(* Logix 5000 project; controller HaileeRenkersACIM5030ProjectFinalVersion vendor 1 type 14 code 54 rev 20.12; software revision 20.01 *)

TASK MainTask (continuous, watchdog 500 ms) : MainProgram

MODULES
   Local : vendor 1 type 14 code 54 (ICP 0, rev 20.12)
      DCinputmodule : 1756-IB16 (ICP 1, rev 3.3, Input RPI 20 ms)   // inputmodule for discrete dc inputs
      outputrelay : 1756-OW16I (ICP 2, rev 3.2, Output RPI 20 ms)   // outputrelay
      inputcardslot3 : 1756-IF8 (ICP 3, rev 1.5, Input RPI 100 ms)
      highspeedcounter : 1756-HSC (ICP 6, rev 3.4, Output RPI 2 ms)
      Ethernet : 1756-ENBT (ICP 7, Ethernet 142.232.195.220, rev 4.8)
         Powerflex : vendor 1 type 123 code 50 (Ethernet 142.232.195.234, rev 5.1, Output RPI 20 ms)
             : vendor 1 type 123 code 8192 (DPI 5, rev 4.2)
             : vendor 1 type 123 code 1535 (DPI 3, rev 6.1)
END_MODULES

VAR_GLOBAL   (* controller tags *)
   AirPressure : ALIAS FOR Local:3:I.Ch0Data;
   AutoKick1 : BOOL;
   AutoKick2 : BOOL;
   AutoKick3 : BOOL;
   AutoKick4 : BOOL;
   Bit_Shift_Oneshot : BOOL;
   Boards_array : DINT[32];
   Control_for_boards : CONTROL := (LEN := 160);
   DriveForward : ALIAS FOR Powerflex:O.DriveLogicRslt_Forward;
   DriveFrequency : ALIAS FOR Powerflex:O.CommandedFreq;
   DriveReverse : ALIAS FOR Powerflex:O.DriveLogicRslt_Reverse;
   DriveStart : ALIAS FOR Powerflex:O.DriveLogicRslt_Start;
   DriveStop : ALIAS FOR Powerflex:O.DriveLogicRslt_Stop;
   FreqHolder : INT;
   HSC_Channel_A : ALIAS FOR Local:6:I.PresentValue[1];
   Increment_OS : BOOL;
   JoystickForward : ALIAS FOR Local:1:I.Data.10;
   Joystickreverse : ALIAS FOR Local:1:I.Data.11;
   Kicker1Button : ALIAS FOR Local:1:I.Data.3;
   Kicker1Solenoid : ALIAS FOR Local:2:O.Data.2;
   Kicker2Button : ALIAS FOR Local:1:I.Data.4;
   Kicker2Solenoid : ALIAS FOR Local:2:O.Data.3;
   Kicker3Button : ALIAS FOR Local:1:I.Data.5;
   Kicker3Solenoid : ALIAS FOR Local:2:O.Data.4;
   Kicker4Button : ALIAS FOR Local:1:I.Data.6;
   Kicker4Solenoid : ALIAS FOR Local:2:O.Data.5;
   Manual_button_PB : ALIAS FOR Local:1:I.Data.9;
   osf_timer : BOOL;
   osf_unlatch : BOOL;
   Photoeye1 : ALIAS FOR Local:1:I.Data.7;
   photoeye1ONS : BOOL;
   Photoeye2 : ALIAS FOR Local:1:I.Data.8;
   PRESSURELIVE : BOOL;
   PSISig : ALIAS FOR Local:1:I.Data.0;
   RPMDisplay : INT;
   RPMplaceholder : INT;
   RPMRatedSpeed : INT;
   RPMSlipHolder : INT;
   Scan_and_sort_light : ALIAS FOR Local:2:O.Data.0;
   Slow_belt_timer : TIMER := (PRE := 7500);
   slow_latch : BOOL;
   STARTPB : ALIAS FOR Local:1:I.Data.1;
   STOPPB : ALIAS FOR Local:1:I.Data.2;
   VFD_OK : ALIAS FOR Local:1:I.Data.12;
   VFD_STATUS_LIGHT : ALIAS FOR Local:2:O.Data.1;
END_VAR

PROGRAM MainProgram   (* main routine MainRoutine *)
VAR
   AirPressureHMI : DINT;
   ALARM_PSI_BOOL : BOOL;
   ALARM_PSI_INT : DINT;
   Auto : BOOL;
   JoystickForward_HMI : BOOL;
   Joystickreverse_HMI : BOOL;
   Kicker1_from_HMI : BOOL;
   Kicker2_from_HMI : BOOL;
   Kicker3_from_HMI : BOOL;
   Kicker4_from_HMI : BOOL;
   Manual : BOOL;
   ManualFrequency : INT;
   ManualOut : BOOL;
   ManualPercent : DINT;
   Photoeye1_MHI : BOOL;
   Photoeye2_MHI : BOOL;
   PSIALARM : BOOL;
   RPM_MOTOR_HMI : INT;
   Solenoid1_HMI : BOOL;
   Solenoid2_HMI : BOOL;
   Solenoid3_HMI : BOOL;
   Solenoid4_HMI : BOOL;
   StartPB_HMI : BOOL;
   StopPB_HMI : BOOL;
   VFD_FAULT_HMI : BOOL;
END_VAR

ROUTINE MainRoutine   (* ladder *)
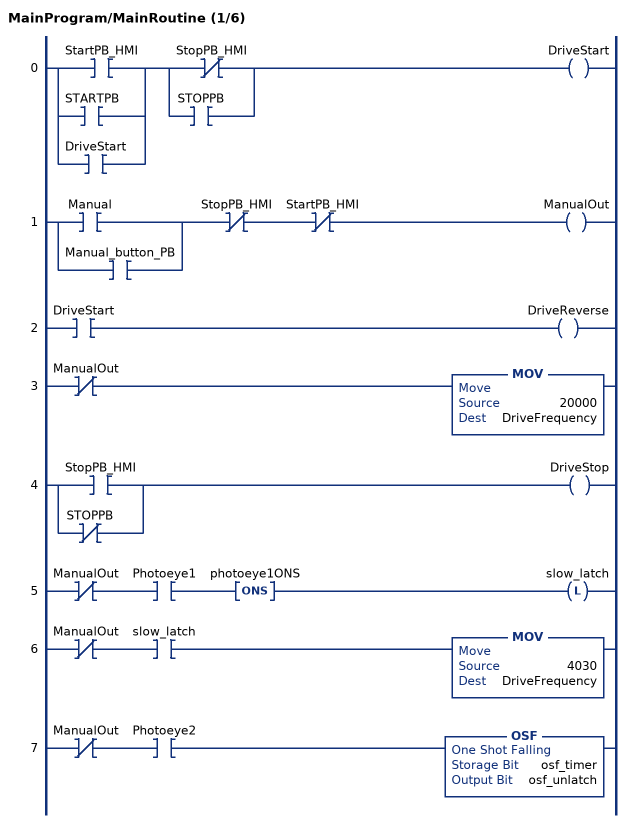
   0: [XIC(StartPB_HMI) ,XIC(STARTPB) ,XIC(DriveStart) ][XIO(StopPB_HMI) ,XIC(STOPPB) ]OTE(DriveStart);
   1: [XIC(Manual) ,XIC(Manual_button_PB) ]XIO(StopPB_HMI)XIO(StartPB_HMI)OTE(ManualOut);
   2: XIC(DriveStart)OTE(DriveReverse);
   3: XIO(ManualOut)MOV(20000,DriveFrequency);
   4: [XIC(StopPB_HMI) ,XIO(STOPPB) ]OTE(DriveStop);
   5: XIO(ManualOut)XIC(Photoeye1)ONS(photoeye1ONS)OTL(slow_latch);
   6: XIO(ManualOut)XIC(slow_latch)MOV(4030,DriveFrequency);
   7: XIO(ManualOut)XIC(Photoeye2)OSF(osf_timer,osf_unlatch);
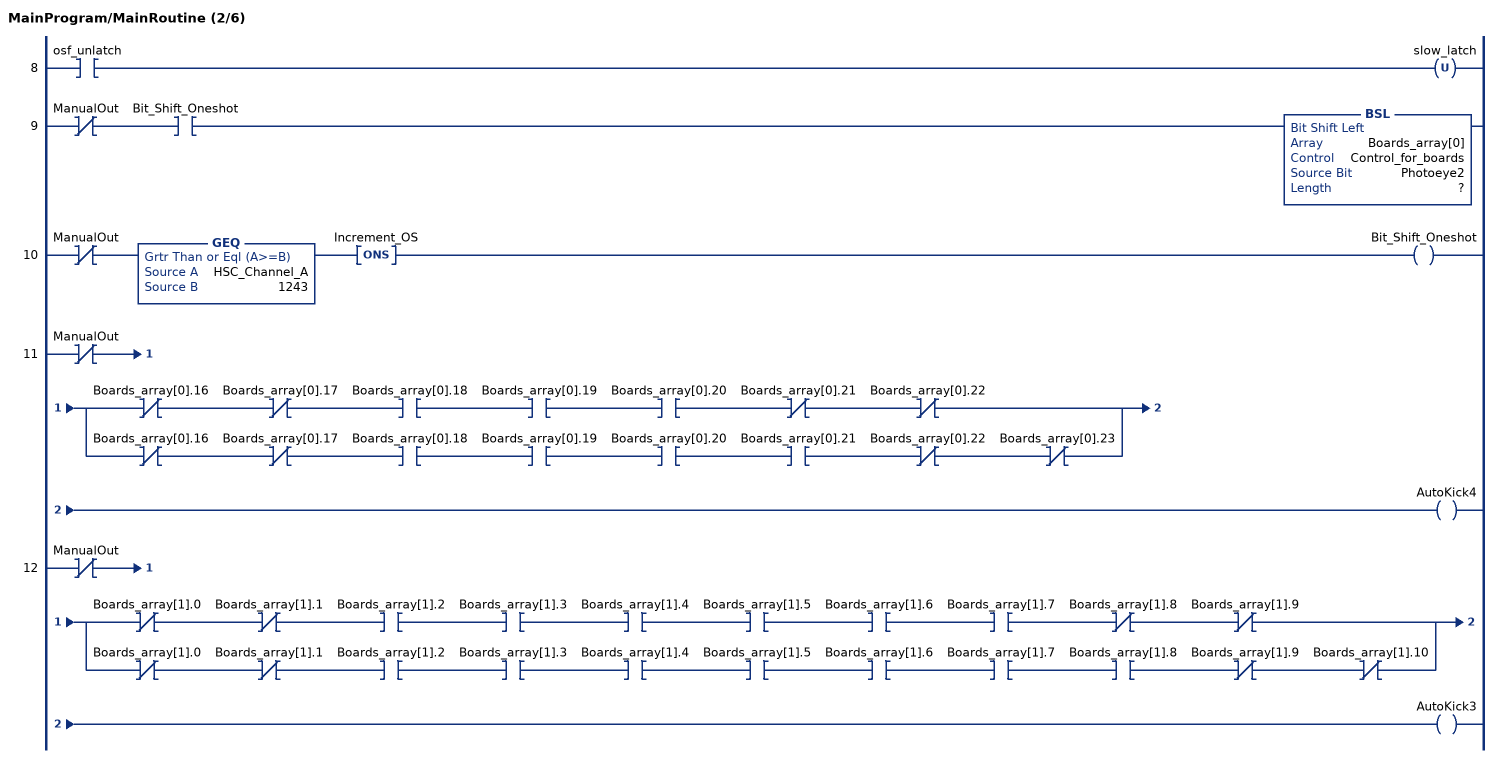
   8: XIC(osf_unlatch)OTU(slow_latch);
   9: XIO(ManualOut)XIC(Bit_Shift_Oneshot)BSL(Boards_array[0],Control_for_boards,Photoeye2,?);
   10: XIO(ManualOut)GEQ(HSC_Channel_A,1243)ONS(Increment_OS)OTE(Bit_Shift_Oneshot);
   11: XIO(ManualOut)[XIO(Boards_array[0].16) XIO(Boards_array[0].17) XIC(Boards_array[0].18) XIC(Boards_array[0].19) XIC(Boards_array[0].20) XIO(Boards_array[0].21) XIO(Boards_array[0].22) ,XIO(Boards_array[0].16) XIO(Boards_array[0].17) XIC(Boards_array[0].18) XIC(Boards_array[0].19) XIC(Boards_array[0].20) XIC(Boards_array[0].21) XIO(Boards_array[0].22) XIO(Boards_array[0].23) ]OTE(AutoKick4);
   12: XIO(ManualOut)[XIO(Boards_array[1].0) XIO(Boards_array[1].1) XIC(Boards_array[1].2) XIC(Boards_array[1].3) XIC(Boards_array[1].4) XIC(Boards_array[1].5) XIC(Boards_array[1].6) XIC(Boards_array[1].7) XIO(Boards_array[1].8) XIO(Boards_array[1].9) ,XIO(Boards_array[1].0) XIO(Boards_array[1].1) XIC(Boards_array[1].2) XIC(Boards_array[1].3) XIC(Boards_array[1].4) XIC(Boards_array[1].5) XIC(Boards_array[1].6) XIC(Boards_array[1].7) XIC(Boards_array[1].8) XIO(Boards_array[1].9) XIO(Boards_array[1].10) ]OTE(AutoKick3);
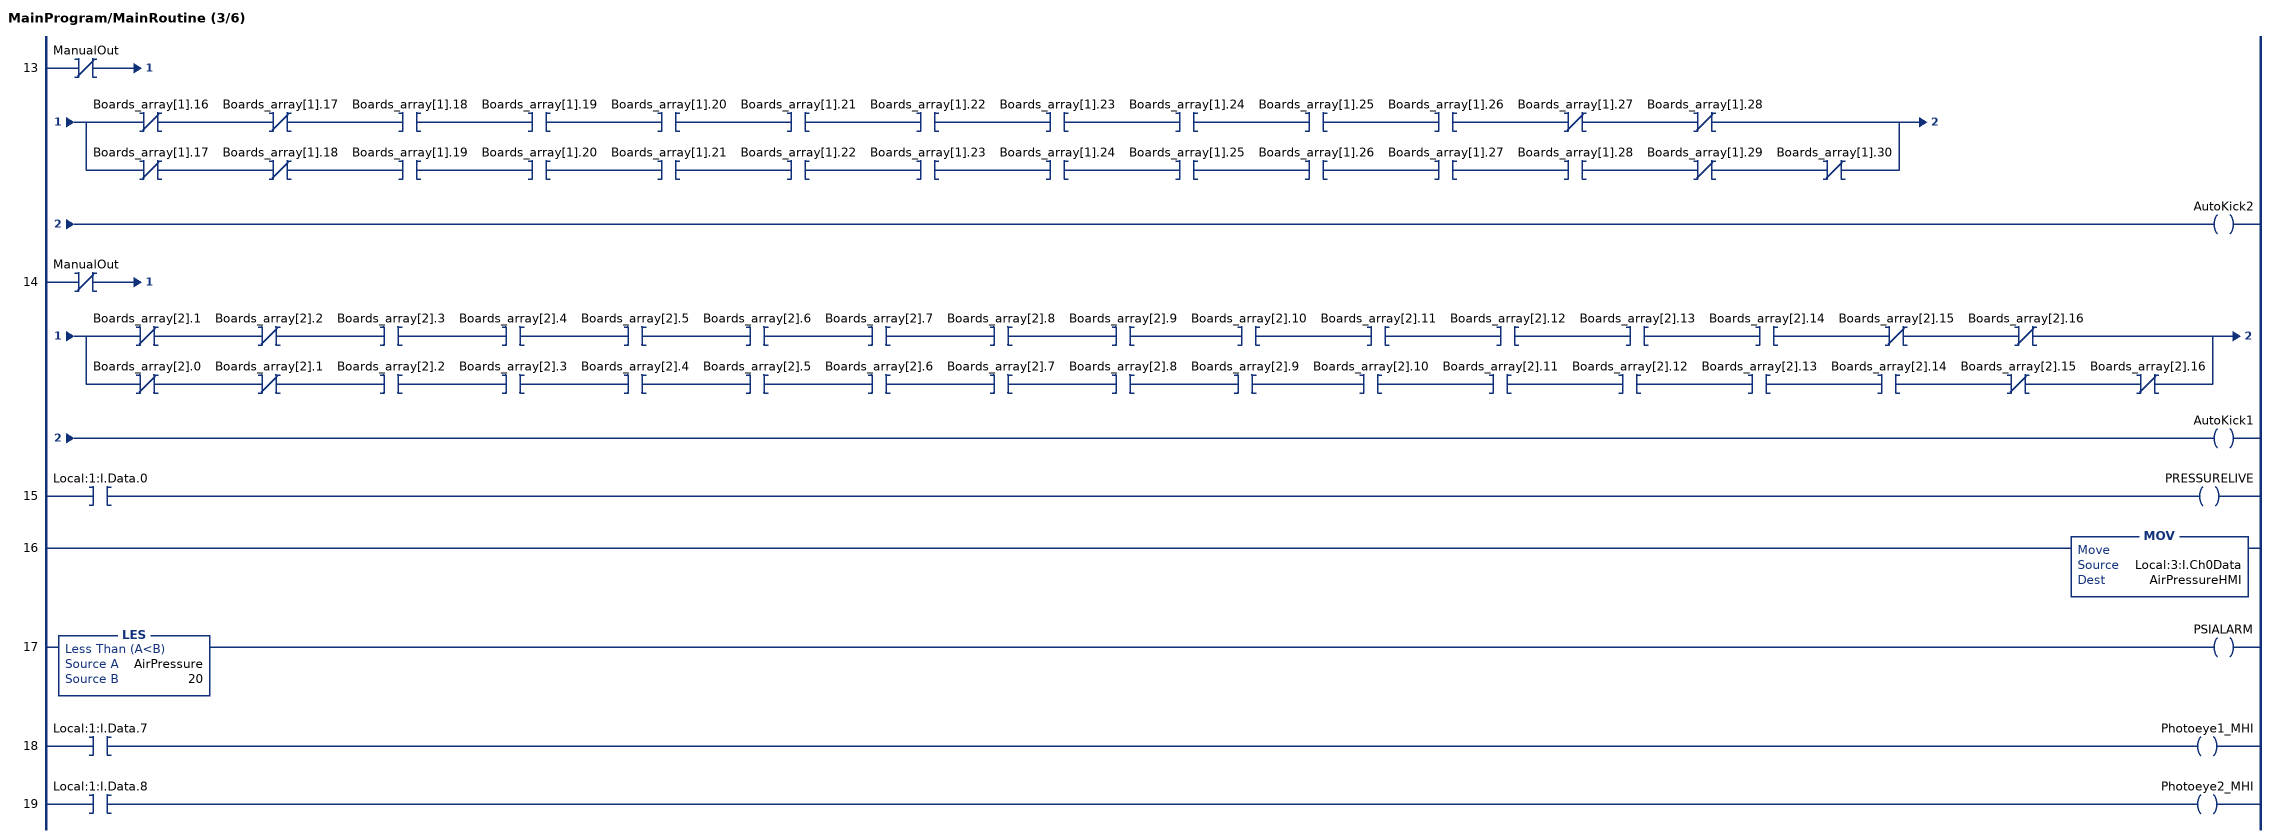
   13: XIO(ManualOut)[XIO(Boards_array[1].16) XIO(Boards_array[1].17) XIC(Boards_array[1].18) XIC(Boards_array[1].19) XIC(Boards_array[1].20) XIC(Boards_array[1].21) XIC(Boards_array[1].22) XIC(Boards_array[1].23) XIC(Boards_array[1].24) XIC(Boards_array[1].25) XIC(Boards_array[1].26) XIO(Boards_array[1].27) XIO(Boards_array[1].28) ,XIO(Boards_array[1].17) XIO(Boards_array[1].18) XIC(Boards_array[1].19) XIC(Boards_array[1].20) XIC(Boards_array[1].21) XIC(Boards_array[1].22) XIC(Boards_array[1].23) XIC(Boards_array[1].24) XIC(Boards_array[1].25) XIC(Boards_array[1].26) XIC(Boards_array[1].27) XIC(Boards_array[1].28) XIO(Boards_array[1].29) XIO(Boards_array[1].30) ]OTE(AutoKick2);
   14: XIO(ManualOut)[XIO(Boards_array[2].1) XIO(Boards_array[2].2) XIC(Boards_array[2].3) XIC(Boards_array[2].4) XIC(Boards_array[2].5) XIC(Boards_array[2].6) XIC(Boards_array[2].7) XIC(Boards_array[2].8) XIC(Boards_array[2].9) XIC(Boards_array[2].10) XIC(Boards_array[2].11) XIC(Boards_array[2].12) XIC(Boards_array[2].13) XIC(Boards_array[2].14) XIO(Boards_array[2].15) XIO(Boards_array[2].16) ,XIO(Boards_array[2].0) XIO(Boards_array[2].1) XIC(Boards_array[2].2) XIC(Boards_array[2].3) XIC(Boards_array[2].4) XIC(Boards_array[2].5) XIC(Boards_array[2].6) XIC(Boards_array[2].7) XIC(Boards_array[2].8) XIC(Boards_array[2].9) XIC(Boards_array[2].10) XIC(Boards_array[2].11) XIC(Boards_array[2].12) XIC(Boards_array[2].13) XIC(Boards_array[2].14) XIO(Boards_array[2].15) XIO(Boards_array[2].16) ]OTE(AutoKick1);
   15: XIC(Local:1:I.Data.0)OTE(PRESSURELIVE);
   16: MOV(Local:3:I.Ch0Data,AirPressureHMI);
   17: LES(AirPressure,20)OTE(PSIALARM);
   18: XIC(Local:1:I.Data.7)OTE(Photoeye1_MHI);
   19: XIC(Local:1:I.Data.8)OTE(Photoeye2_MHI);
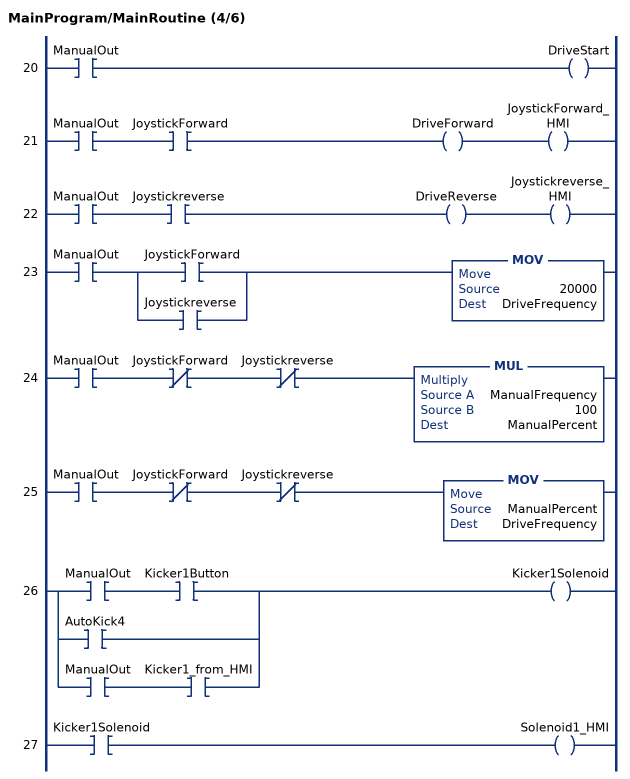
   20: XIC(ManualOut)OTE(DriveStart);
   21: XIC(ManualOut)XIC(JoystickForward)OTE(DriveForward)OTE(JoystickForward_HMI);
   22: XIC(ManualOut)XIC(Joystickreverse)OTE(DriveReverse)OTE(Joystickreverse_HMI);
   23: XIC(ManualOut)[XIC(JoystickForward) ,XIC(Joystickreverse) ]MOV(20000,DriveFrequency);
   24: XIC(ManualOut)XIO(JoystickForward)XIO(Joystickreverse)MUL(ManualFrequency,100,ManualPercent);
   25: XIC(ManualOut)XIO(JoystickForward)XIO(Joystickreverse)MOV(ManualPercent,DriveFrequency);
   26: [XIC(ManualOut) XIC(Kicker1Button) ,XIC(AutoKick4) ,XIC(ManualOut) XIC(Kicker1_from_HMI) ]OTE(Kicker1Solenoid);
   27: XIC(Kicker1Solenoid)OTE(Solenoid1_HMI);
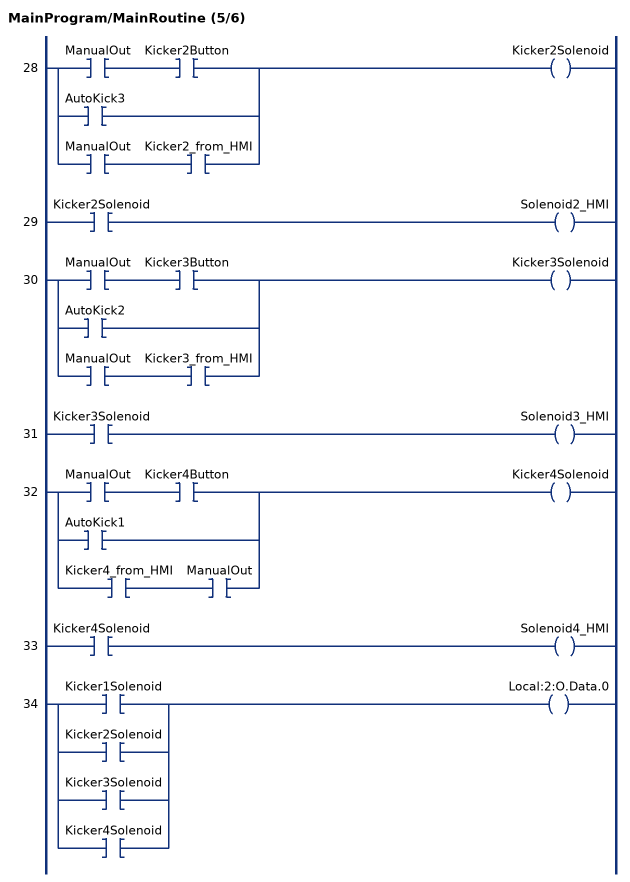
   28: [XIC(ManualOut) XIC(Kicker2Button) ,XIC(AutoKick3) ,XIC(ManualOut) XIC(Kicker2_from_HMI) ]OTE(Kicker2Solenoid);
   29: XIC(Kicker2Solenoid)OTE(Solenoid2_HMI);
   30: [XIC(ManualOut) XIC(Kicker3Button) ,XIC(AutoKick2) ,XIC(ManualOut) XIC(Kicker3_from_HMI) ]OTE(Kicker3Solenoid);
   31: XIC(Kicker3Solenoid)OTE(Solenoid3_HMI);
   32: [XIC(ManualOut) XIC(Kicker4Button) ,XIC(AutoKick1) ,XIC(Kicker4_from_HMI) XIC(ManualOut) ]OTE(Kicker4Solenoid);
   33: XIC(Kicker4Solenoid)OTE(Solenoid4_HMI);
   34: [XIC(Kicker1Solenoid) ,XIC(Kicker2Solenoid) ,XIC(Kicker3Solenoid) ,XIC(Kicker4Solenoid) ]OTE(Local:2:O.Data.0);
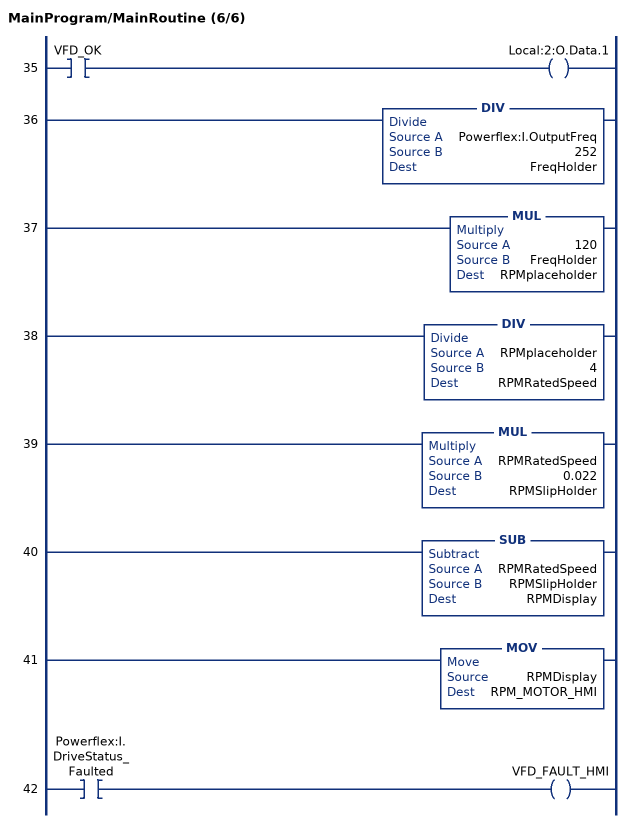
   35: XIC(VFD_OK)OTE(Local:2:O.Data.1);
   36: DIV(Powerflex:I.OutputFreq,252,FreqHolder);
   37: MUL(120,FreqHolder,RPMplaceholder);
   38: DIV(RPMplaceholder,4,RPMRatedSpeed);
   39: MUL(RPMRatedSpeed,0.022,RPMSlipHolder);
   40: SUB(RPMRatedSpeed,RPMSlipHolder,RPMDisplay);
   41: MOV(RPMDisplay,RPM_MOTOR_HMI);
   42: XIC(Powerflex:I.DriveStatus_Faulted)OTE(VFD_FAULT_HMI);
END_ROUTINE
END_PROGRAM
